# B&R Automation Studio project spro-4-rd-pendulum-main
Automation Studio 4.9

## Configuration Config1

CPU X20CP1382, AutomationRuntime H4.83, Build 4.1.2, Vc V4.73.2

### IoMap.iom - X20CP1382/IoMap.iom
```iecst
VAR_CONFIG
	::I_pos_pendulum AT %ID."X2".Counter01Value;
	::I_pos_cart AT %ID."X2".Counter02Value;
	::reset_cart_position AT %QX."X2".Counter02Reset;
	::reset_pendulum_position AT %QX."X2".Counter01Reset;
	::I_endstop_negative AT %IX."X2".DigitalInput09;
	::I_endstop_positive AT %IX."X2".DigitalInput10;
	::I_drive_active AT %IX."X2".DigitalInput08;
	::I_drive_no_fault AT %IX."X2".DigitalInput07;
	::Q_vel_cart AT %QW."X20AO2622".AnalogOutput01;
	::Q_drive_enable AT %QX."X3".DigitalOutput01;
	::Q_drive_operating_mode AT %QX."X3".DigitalOutput02;
	::Q_drive_faultreset AT %QX."X3".DigitalOutput03;
	::SI_estop_A AT %IX."X1".DigitalInput01;
	::SI_estop_B AT %IX."X1".DigitalInput02;
	::SI_reset_btn AT %IX."X1".DigitalInput03;
	::Q_reset_LED AT %QX."X3".DigitalOutput05;
END_VAR
```

## Logical view

### Global.var
```iecst
VAR
	SI_estop_B : BOOL;
	SI_estop_A : BOOL;
	SI_reset_btn : BOOL;
	I_drive_active : BOOL;
	I_drive_no_fault : BOOL;
	I_endstop_negative : BOOL;
	I_endstop_positive : BOOL;
	I_pos_cart : DINT;
	I_pos_pendulum : DINT;
	Q_drive_enable : BOOL;
	Q_drive_faultreset : BOOL;
	Q_drive_operating_mode : BOOL;
	Q_vel_cart : INT;
	Q_reset_LED : BOOL;
	reset_cart_position : BOOL;
	reset_pendulum_position : BOOL;
	A : ARRAY[0..3,0..3] OF REAL := [1.0,0.009535,0.0000575,0.0000002737,0.0,0.9085,-0.01132,0.00003438,0.0,0.001945,1.002,0.009989,0.0,0.3829,0.4582,0.9986];
	B : ARRAY[0..3] OF REAL := [0.001859,0.366,-0.007782,-1.531];
	K : ARRAY[0..3] OF REAL := [-9.97788845498053,-4.33797239803683,-8.31962221505295,-1.27391028745717];
	u : REAL;
	x : ARRAY[0..3] OF REAL;
	x_out : ARRAY[0..3] OF REAL;
END_VAR
```

### Types.typ
```iecst
TYPE
	Position_case :
		(
		position0,
		position1,
		position2,
		position3,
		position4,
		position5,
		position6,
		position7,
		position8,
		position9,
		position10
		);
END_TYPE
```
